// TIA Portal V16 export
// export: Created 2024-09-05T17:40:14.3376251Z, ExportSetting WithDefaults, DisplayName Totally Integrated Automation Portal, DisplayVersion V16 Update 6, DisplayName TIA Portal Version Control Interface, DisplayVersion V16 Update 2, DisplayName TIA Portal Openness, DisplayVersion V16 Update 6, DisplayName STEP 7 Professional, DisplayVersion V16 Update 6, DisplayName STEP 7 Safety, DisplayVersion V16, DisplayName WinCC Advanced, DisplayVersion V16 Update 6
TYPE "UDT_Robot"
// stored: IsFailsafeCompliant false
   STRUCT
      StartReq : Bool;
      StartAllowed : Bool;
      Started : Bool;
      Job : Struct
         JobNr : Byte;
         Start : Bool;
         Done : Bool;
      END_STRUCT;
   END_STRUCT;
END_TYPE
